(* PLC project Tc2_Utilities.FB_FileTime64ToTzSpecificLocalTime Demo, tc3-libraries-kb TwinCAT 3.1 *)
(* stored: creationDateTime 2026-05-11T00:00:00, modificationDateTime 2026-05-11T00:00:00 *)

PROGRAM P_Demo_FB_FileTime64ToTzSpecificLocalTime
  VAR
    fbFB_FileTime64ToTzSpecificLocalTime : FB_FileTime64ToTzSpecificLocalTime;  (* FB_FileTime64ToTzSpecificLocalTime 实例 *)
    bConv : BOOL := FALSE;
    stTz : TIME_ZONE_INFORMATION;
    stFt : T_ULARGE_INTEGER;
    stLocalOut : TIMESTRUCT;
  END_VAR

// =============================================================================
// 场景：读文件修改 FileTime 转本地。
// 价值：封装 epoch + 时区计算。
// 验证：给 stFt 填一个典型 FileTime（如 130428000000000000，约 2014 年），转换后 stLocalOut 应为合理本地时间。
// 验证步骤：
//   1. 右键 PLC 项目 → Import PLCopenXML → 选本文件
//   2. 引用 Tc2_Utilities（References → Add library）
//   3. 编译 → 登录 → 运行；按上方『验证』行的指示在线写值观察
// =============================================================================

fbFB_FileTime64ToTzSpecificLocalTime(
    tzInfo := stTz, bExecute := bConv, stFileTime := stFt,
    stLocal => stLocalOut
);
END_PROGRAM
